PROGRAM LadderLogicBottleChecker
VAR
	{attribute 'OPC.UA.DA' := '1'}
	ProximitySensor: BOOL;
	{attribute 'OPC.UA.DA' := '1'}
	BottleDetected: BOOL;
	ProximityTimer: TON;
	{attribute 'OPC.UA.DA' := '1'}
	EjectBottle: BOOL;
	{attribute 'OPC.UA.DA' := '1'}
	EjectRelay: BOOL;
	EjectionTimer: TON;
	{attribute 'OPC.UA.DA' := '1'}
	ExitScript: BOOL;
	
	SessionCounter: CTU;
	{attribute 'OPC.UA.DA' := '1'}
	sessionNumber: INT;
	RejectFlag: BOOL;
	AcceptFlag: BOOL;
END_VAR
VAR // added by the converter: edge detectors and wires of the graphical bodies
    _rt1 : R_TRIG;
END_VAR

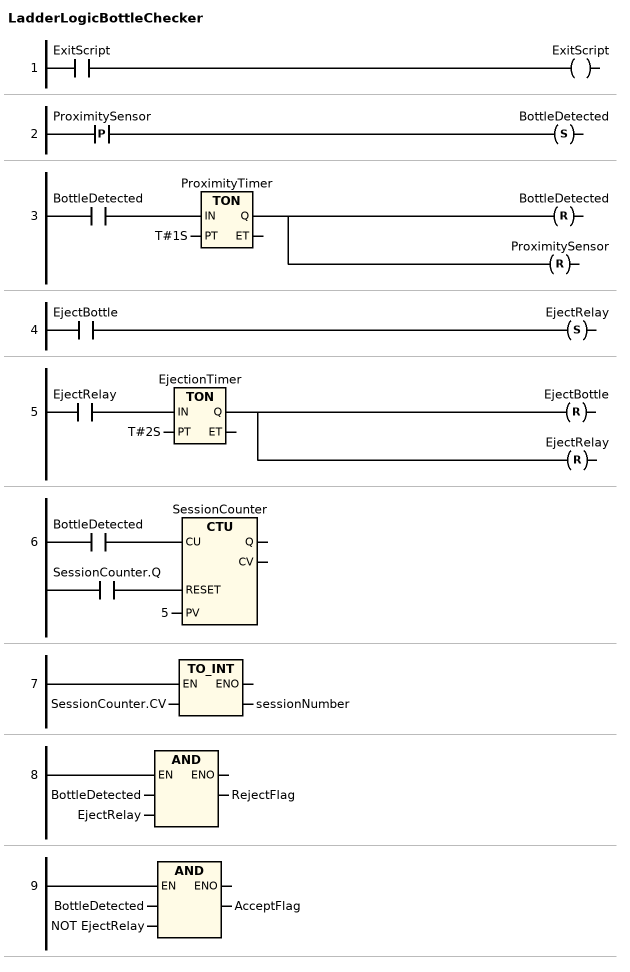
// NETWORK 1
ExitScript := ExitScript;

// NETWORK 2
_rt1(CLK := ProximitySensor);
BottleDetected S= _rt1.Q;

// NETWORK 3
ProximityTimer(IN := BottleDetected, PT := T#1S); // TON
BottleDetected R= ProximityTimer.Q;
ProximitySensor R= ProximityTimer.Q;

// NETWORK 4
EjectRelay S= EjectBottle;

// NETWORK 5
EjectionTimer(IN := EjectRelay, PT := T#2S); // TON
EjectBottle R= EjectionTimer.Q;
EjectRelay R= EjectionTimer.Q;

// NETWORK 6
SessionCounter(CU := BottleDetected, RESET := SessionCounter.Q, PV := 5); // CTU

// NETWORK 7
sessionNumber := TO_INT(SessionCounter.CV);

// NETWORK 8
RejectFlag := BottleDetected AND EjectRelay;

// NETWORK 9
AcceptFlag := BottleDetected AND (NOT EjectRelay);

END_PROGRAM

(* stored: Version 1.1.0.1, ProductVersion 3.1.4026.8
   POU LadderLogicBottleChecker: Id {a95e250c-788e-4011-b630-ffb36cc19941}, SpecialFunc None *)
